(* CoDeSys 2.3 export: LOCKMODE.EXP *)

(* POU Global/LockMode, ST *)
FUNCTION_BLOCK LockMode
VAR_INPUT
END_VAR
VAR_OUTPUT
END_VAR
VAR
	Button: Button;
	allShaders: ARRAY [0..6] OF POINTER TO Shader;
	i: INT;
END_VAR
button(input:=H9_2c);

allShaders[0]:= ADR(shader_kuchnia);
allShaders[1]:= ADR(shader_taras);
allShaders[2]:= ADR(shader_kominek);
allShaders[3]:= ADR(shader_gabinet);
allShaders[4]:= ADR(shader_sypialnia);
allShaders[5]:= ADR(shader_lazienka);
allShaders[6]:= ADR(shader_kotlownia); (* close only *)

IF button.longPressed THEN
	FOR i := 0 TO 6 DO
		allShaders[i]^.closeImpulse := 1;
	END_FOR
END_IF

IF button.fallingEdge THEN
	FOR i := 0 TO 5 DO
		allShaders[i]^.openImpulse := 1;
	END_FOR
END_IF
END_FUNCTION_BLOCK
